FUNCTION F_UpdateFunc_REF : REAL
VAR_INPUT
	bUpdateValue : BOOL;
	fNewValue : REAL; 
	stMotorParameter : REFERENCE TO ST_MotorParams; 
END_VAR
VAR
END_VAR

IF bUpdateValue THEN
	stMotorParameter.fMaxSpeed := fNewValue; 
	ELSE
		stMotorParameter.fMaxSpeed := stMotorParameter.fMaxSpeed; 

END_IF;

END_FUNCTION

(* stored: Version 1.1.0.1, ProductVersion 3.1.4024.12
   POU F_UpdateFunc_REF: Id {35956870-633c-4141-a88e-028e67051681}, SpecialFunc None *)
